# EPICS autosave request: apps/wf2rootApp/Db/wf2root_settings.req
#
# wf2root_settings.req - autosave, waveform -> root file
#
# Author: Wesley Moore (wmoore@jlab.org)
# Date:   Mar 2016
#
$(P)ctrl:daq_state
$(P)ctrl:file_limit
